(* IEC 61131-3 sources: crb-codesys/retrieval/output/codesys_repo/plc_hello_mixing_tank/PRG, 2 files *)

(* ---- main.st ---- *)
PROGRAM main
VAR
	///模式控制器
	fbModeController		:	FB_ModeController;
	///手动控制功能块
	fbManualControl			:	FB_ManualControl;
	///自动序列控制功能块
	fbAutoSequence			:	FB_AutoSequence;

	///当前运行模式
	vMode					:	MODES;
END_VAR
(*Functional description:
There are two ways of operation:
	- Manual
	- Automatic
Manual:
	- Operator is able to operate each valve manually
	- Operator is able to operate the mixer motor manually
	- Overfill protections are disabled
	- Operator is able to put the system to auto

Automatic:
	- Program will automatically control the valves and the mixing motor if system is in auto
	- If the tanks level is undefined it assumes draining state
	- In draining state, drains the tank until LS02 activates (tank is empty)
	- When tank is empty, it activates the medium 1 and 2 valves, closes the drain valve and the tank is filling up
	- Filling state is until LS01 is activated (Tank is full)
	- Then the mixer motor is mixing for 10 seconds
	- After mixing is completed, drain the whole contents
	- Repeats as long as auto is activated

HMI Requirements:
	- Manual / Auto needs to be correctly controlled and displayed
	- If manual, clicking on devices activates or stops them
	- If auto, clicking is not doing anything
	- If auto, system is counting number of cycles completed
	- Devices must clearly display if they are activated or deactivated*)

// ========== 模式控制 ==========
fbModeController(
	bSetToAuto := HMI.SetToAuto,
	bSetToManual := HMI.SetToManual
);
vMode := fbModeController.eCurrentMode;

// 模式切换时，复位HMI命令
IF fbModeController.bModeChanged THEN
	HMI.SetToAuto := FALSE;
	HMI.SetToManual := FALSE;
END_IF

// ========== 控制逻辑 ==========
CASE vMode OF
	MODES.MANUAL: (*手动模式*)
		// 使用手动控制功能块
		fbManualControl(
			bMixerRunCmd := HMI.MixerRunCmd,
			bMixerStopCmd := HMI.MixerStopCmd,
			bMedium1OpenCmd := HMI.Medium1OpenCmd,
			bMedium1CloseCmd := HMI.Medium1CloseCmd,
			bMedium2OpenCmd := HMI.Medium2OpenCmd,
			bMedium2CloseCmd := HMI.Medium2CloseCmd,
			bDrainOpenCmd := HMI.DrainOpenCmd,
			bDrainCloseCmd := HMI.DrainCloseCmd,
			bMixerRunning := IO.xDI_M1_MixerMotorRunning,
			bMedium1Opened := IO.xDI_VV01_Medium1_Opened,
			bMedium2Opened := IO.xDI_VV02_Medium2_Opened,
			bDrainOpened := IO.xDI_VV03_TankDrain_Opened
		);

		// 输出到IO
		IO.xDO_M1_MixerMotorRunCmd := fbManualControl.bMixerRunCmdOut;
		IO.xDO_VV01_Medium1_OpenCmd := fbManualControl.bMedium1OpenCmdOut;
		IO.xDO_VV02_Medium2_OpenCmd := fbManualControl.bMedium2OpenCmdOut;
		IO.xDO_VV03_TankDrain_OpenCmd := fbManualControl.bDrainOpenCmdOut;

		// 自动序列禁用
		fbAutoSequence(bEnable := FALSE);

	MODES.AUTO: (*自动模式*)
		// 使用自动序列功能块
		fbAutoSequence(
			bEnable := TRUE,
			bReset := fbModeController.bModeChanged,
			bTankLevelFull := IO.xDI_LS01_TankLevelFull,
			bTankLevelEmpty := IO.xDI_LS02_TankLevelEmpty,
			bMixerRunning := IO.xDI_M1_MixerMotorRunning,
			bMedium1Opened := IO.xDI_VV01_Medium1_Opened,
			bMedium2Opened := IO.xDI_VV02_Medium2_Opened,
			bDrainOpened := IO.xDI_VV03_TankDrain_Opened,
			tMixingDuration := T#10S
		);

		// 输出到IO
		IO.xDO_M1_MixerMotorRunCmd := fbAutoSequence.bMixerRunCmd;
		IO.xDO_VV01_Medium1_OpenCmd := fbAutoSequence.bMedium1OpenCmd;
		IO.xDO_VV02_Medium2_OpenCmd := fbAutoSequence.bMedium2OpenCmd;
		IO.xDO_VV03_TankDrain_OpenCmd := fbAutoSequence.bDrainOpenCmd;

		// 更新循环计数
		HMI.CyclesCompleted := fbAutoSequence.nCyclesCompleted;
END_CASE

// ========== HMI命令复位 ==========
F_ResetDeviceCommands(
	bMixerRunCmd := HMI.MixerRunCmd,
	bMixerStopCmd := HMI.MixerStopCmd,
	bMedium1OpenCmd := HMI.Medium1OpenCmd,
	bMedium1CloseCmd := HMI.Medium1CloseCmd,
	bMedium2OpenCmd := HMI.Medium2OpenCmd,
	bMedium2CloseCmd := HMI.Medium2CloseCmd,
	bDrainOpenCmd := HMI.DrainOpenCmd,
	bDrainCloseCmd := HMI.DrainCloseCmd,
	bMixerRunning := IO.xDI_M1_MixerMotorRunning,
	bMedium1Opened := IO.xDI_VV01_Medium1_Opened,
	bMedium2Opened := IO.xDI_VV02_Medium2_Opened,
	bDrainOpened := IO.xDI_VV03_TankDrain_Opened
);

// ========== HMI状态更新 ==========
HMI.MotorRotating := HMI.MotorRotating + 2 * BOOL_TO_REAL(IO.xDI_M1_MixerMotorRunning);
IF HMI.MotorRotating >= 360 THEN
	HMI.MotorRotating := 0;
END_IF
HMI.InAuto := vMode = MODES.AUTO;
HMI.InManual := vMode = MODES.MANUAL;

(* ---- simulator.st ---- *)
PROGRAM simulator
VAR
	///模拟混合电机
	MixerMotor				:	GenericBistableDeviceModel;
	///模拟介质1填充阀门
	MediumValve1			:	GenericBistableDeviceModel;
	///模拟介质2填充阀门
	MediumValve2			:	GenericBistableDeviceModel;
	///模拟排空阀门
	DrainValve				:	GenericBistableDeviceModel;

	///液位模拟器
	fbTankLevelSimulator	:	FB_TankLevelSimulator;

	///当前液位
	vTankLevel				:	REAL;
	///电机旋转角度（HMI用）
	vMotorRotating			:	REAL;
END_VAR

// ========== 电机和阀门模拟 ==========
MixerMotor(
	ActivateCmd := IO.xDO_M1_MixerMotorRunCmd,
	DeactivateCmd := NOT IO.xDO_M1_MixerMotorRunCmd,
	cfgActTime := T#2S,
	cfgDeactTime := T#0S,
	Activated => IO.xDI_M1_MixerMotorRunning
);

MediumValve1(
	ActivateCmd := IO.xDO_VV01_Medium1_OpenCmd,
	DeactivateCmd := NOT IO.xDO_VV01_Medium1_OpenCmd,
	cfgActTime := T#1S,
	cfgDeactTime := T#1S,
	Activated => IO.xDI_VV01_Medium1_Opened
);

MediumValve2(
	ActivateCmd := IO.xDO_VV02_Medium2_OpenCmd,
	DeactivateCmd := NOT IO.xDO_VV02_Medium2_OpenCmd,
	cfgActTime := T#1S,
	cfgDeactTime := T#1S,
	Activated => IO.xDI_VV02_Medium2_Opened
);

DrainValve(
	ActivateCmd := IO.xDO_VV03_TankDrain_OpenCmd,
	DeactivateCmd := NOT IO.xDO_VV03_TankDrain_OpenCmd,
	cfgActTime := T#1S,
	cfgDeactTime := T#1S,
	Activated => IO.xDI_VV03_TankDrain_Opened
);

// ========== 液位模拟 ==========
fbTankLevelSimulator(
	bMedium1Opened := MediumValve1.Activated,
	bMedium2Opened := MediumValve2.Activated,
	bDrainOpened := DrainValve.Activated,
	bReset := FALSE,
	rInitialLevel := 25.0,
	rFillRate1 := 0.1,
	rFillRate2 := 0.1,
	rDrainRate := 0.2,
	rMinLevel := 0.0,
	rMaxLevel := 100.0
);
vTankLevel := fbTankLevelSimulator.rCurrentLevel;

// ========== 液位开关模拟 ==========
F_UpdateLimitSwitches(
	rTankLevel := vTankLevel,
	rFullThreshold := 85.0,
	rEmptyThreshold := 5.0,
	bLevelFull => IO.xDI_LS01_TankLevelFull,
	bLevelEmpty => IO.xDI_LS02_TankLevelEmpty
);

// ========== HMI 电机旋转动画 ==========
vMotorRotating := vMotorRotating + 1 * BOOL_TO_REAL(MixerMotor.Activated);
IF vMotorRotating >= 360 THEN
	vMotorRotating := 0;
END_IF
